// TIA Portal V18 export
TYPE "UDT_nokButtonIO"
// stored: IsFailsafeCompliant false
   STRUCT
      I_Button : Bool;
      O_Led : Bool;
   END_STRUCT;
END_TYPE
